// TIA Portal V20 export
DATA_BLOCK "LocalRecordsBuffer"   // DB256
// stored: MemoryReserve 100, Namespace Unit1
   VAR
      CellData { ExternalAccessible := 'False'; ExternalVisible := 'False'; ExternalWritable := 'False'} : Array[0..9] of "LPFE_typeCellDataLBuffer";
      ModuleData { ExternalAccessible := 'False'; ExternalVisible := 'False'; ExternalWritable := 'False'} : Array[0..9] of "LPFE_typeModuleDataLBuffer";
      SectionData { ExternalAccessible := 'False'; ExternalVisible := 'False'; ExternalWritable := 'False'} : Array[0..9] of "LPFE_typeSectionDataLBuffer";
      ToolingData { ExternalAccessible := 'False'; ExternalVisible := 'False'; ExternalWritable := 'False'} : Array[0..9] of "LPFE_typeTPUTToolingDataLBuffer";
      HistGenericPayload { ExternalAccessible := 'False'; ExternalVisible := 'False'; ExternalWritable := 'False'} : Array[0..9] of "LPFE_typeGenericPayloadLBuffer";
      StatusData { ExternalAccessible := 'False'; ExternalVisible := 'False'; ExternalWritable := 'False'} : Array[0..9] of "LPFE_typeGenericPayloadLBuffer";
   END_VAR
BEGIN
END_DATA_BLOCK
